TYPE ST_LinkVariableNode :
STRUCT
	Name : STRING(255);
	Address : PVOID;
	Size : UDINT;
	DataType : E_ConfigDataType;
	Access : E_VariableAccess;
END_STRUCT
END_TYPE

(* stored: Version 1.1.0.1, ProductVersion 3.1.4026.18
   DUT ST_LinkVariableNode: Id {ee532905-1ee8-4eb8-b63e-912291af2e98} *)
